(* Schneider Machine Expert - Basic project laba2, file version 2.4.0.0 *)
(* ProjectInformations: Name=New project *)

HARDWARE
  Cpu 0: TM221C16T
  Cartridge1 0: TMC2AQ2V
  EthernetConfiguration: NetworkName=M221, IpAllocationMode=FixedAddress, IpAddress=0.0.0.0, SubnetMask=0.0.0.0
  EthernetConfiguration: NetworkName=M221, IpAllocationMode=FixedAddress, IpAddress=0.0.0.0, SubnetMask=0.0.0.0
  SerialLineConfiguration: Baud=Baud19200, Parity=ParityEven, DataBits=DataBits8, StopBits=StopBits1, PhysicalMedium=PhysicalMediumRs485, TransmissionMode=TransmissionModeModbusRtu, SlaveId=1, Addressing=SlaveAddressing
  MastTask: UsePeriodScanMode=false, PeriodScan=100
  FastTask: Period=255
  CpuBehavior: StartingMode=StartAsPreviousState, AutoSaveRamOnEeprom=true, WatchdogPeriod=250

SYMBOLS  (address, symbol, comment, settings)
  %M100     S_IDLE
  %M101     S_LOAD1
  %M102     S_LOAD2
  %M103     S_HEA1
  %M104     S_HEA2
  %M105     S_DWNLD
  %S13      SB_FIRSTRUN  "Indicates the first controller cycle in RUN mode"
  %I0.0     SB1_PUSK
  %I0.1     SB2_STOP
  %I0.2     LS1_LO
  %I0.3     LS2_MD
  %I0.4     LS3_HI
  %Q0.0     LVS1
  %Q0.1     LVS2
  %Q0.2     LVS3
  %IW0.0    TE1  [Type=Type_0_10V, Scope=Scope_Normal, Minimum=0, Maximum=1000]
  %QW0.100  TV1  [Type=Type_0_10V, Scope=Scope_Customized, Minimum=0, Maximum=10000]

POU New POU
  (* SectionNumber=1 *)

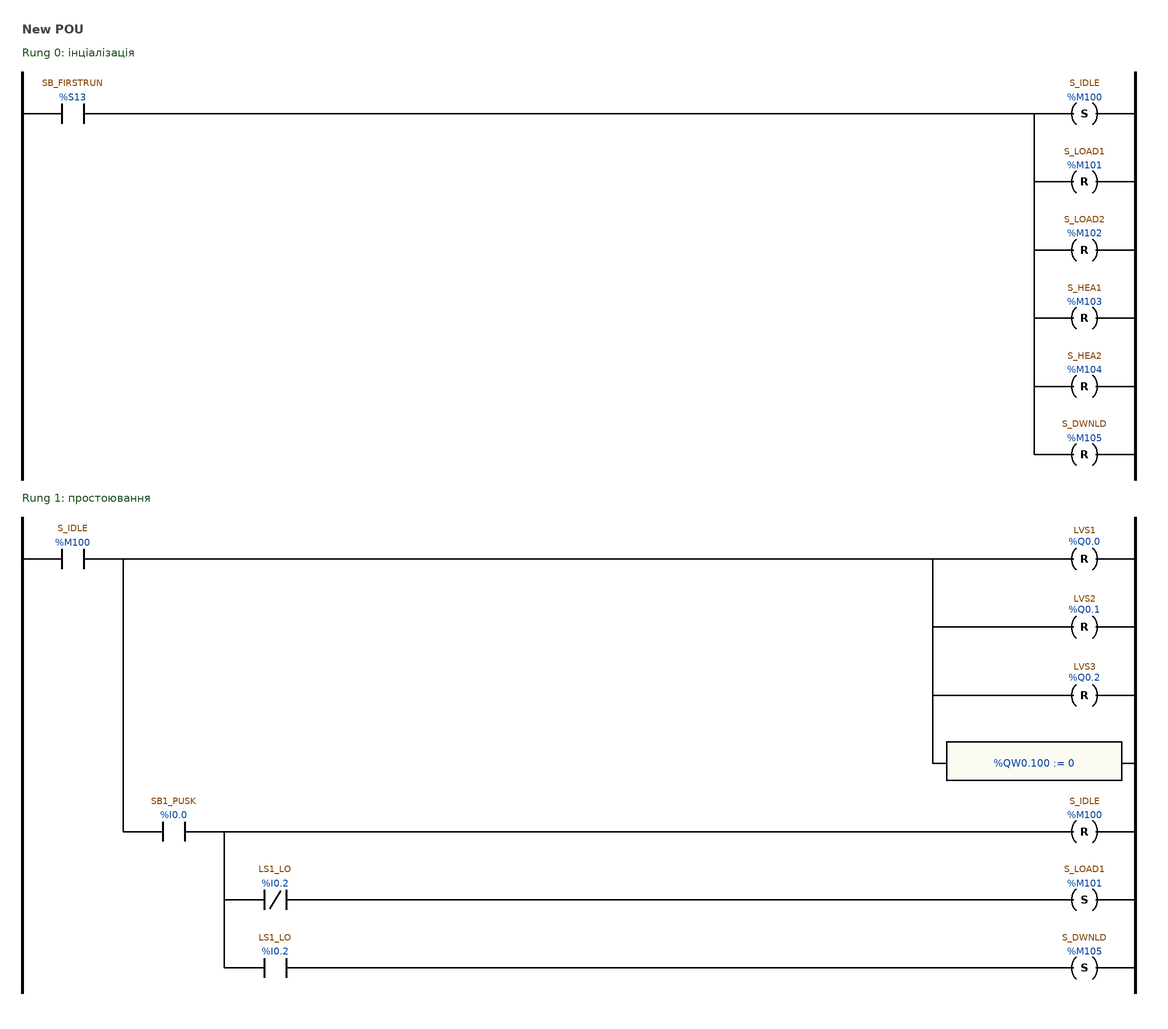

// Rung 0: інціалізація
  LD %S13                 (* SB_FIRSTRUN *)
  S %M100                 (* S_IDLE *)
  R %M101                 (* S_LOAD1 *)
  R %M102                 (* S_LOAD2 *)
  R %M103                 (* S_HEA1 *)
  R %M104                 (* S_HEA2 *)
  R %M105                 (* S_DWNLD *)
  // as ST:
  //   IF SB_FIRSTRUN THEN S_IDLE := TRUE; END_IF;
  //   IF SB_FIRSTRUN THEN S_LOAD1 := FALSE; END_IF;
  //   IF SB_FIRSTRUN THEN S_LOAD2 := FALSE; END_IF;
  //   IF SB_FIRSTRUN THEN S_HEA1 := FALSE; END_IF;
  //   IF SB_FIRSTRUN THEN S_HEA2 := FALSE; END_IF;
  //   IF SB_FIRSTRUN THEN S_DWNLD := FALSE; END_IF;

// Rung 1: простоювання
  LD %M100                (* S_IDLE *)
  MPS
  R %Q0.0                 (* LVS1 *)
  R %Q0.1                 (* LVS2 *)
  R %Q0.2                 (* LVS3 *)
  [ %QW0.100 := 0 ]       (* TV1 *)
  MPP
  AND %I0.0               (* SB1_PUSK *)
  MPS
  R %M100                 (* S_IDLE *)
  MRD
  ANDN %I0.2              (* LS1_LO *)
  S %M101                 (* S_LOAD1 *)
  MPP
  AND %I0.2               (* LS1_LO *)
  S %M105                 (* S_DWNLD *)
  // as ST:
  //   IF S_IDLE THEN LVS1 := FALSE; END_IF;
  //   IF S_IDLE THEN LVS2 := FALSE; END_IF;
  //   IF S_IDLE THEN LVS3 := FALSE; END_IF;
  //   IF S_IDLE THEN TV1 := 0; END_IF;
  //   _t1 := S_IDLE AND SB1_PUSK;
  //   IF _t1 THEN S_IDLE := FALSE; END_IF;
  //   IF _t1 AND NOT LS1_LO THEN S_LOAD1 := TRUE; END_IF;
  //   IF _t1 AND LS1_LO THEN S_DWNLD := TRUE; END_IF;

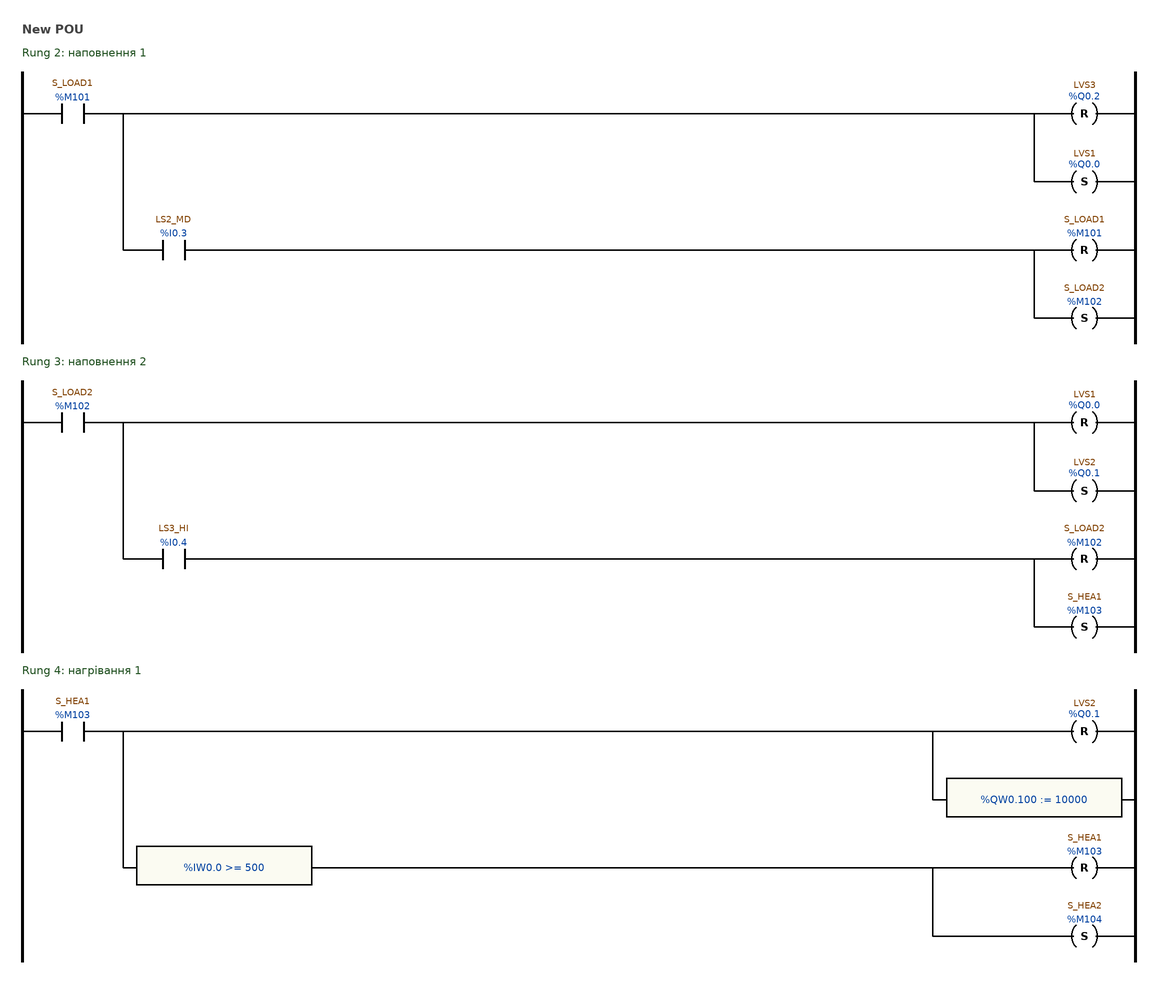

// Rung 2: наповнення 1
  LD %M101                (* S_LOAD1 *)
  MPS
  R %Q0.2                 (* LVS3 *)
  S %Q0.0                 (* LVS1 *)
  MPP
  AND %I0.3               (* LS2_MD *)
  R %M101                 (* S_LOAD1 *)
  S %M102                 (* S_LOAD2 *)
  // as ST:
  //   IF S_LOAD1 THEN LVS3 := FALSE; END_IF;
  //   IF S_LOAD1 THEN LVS1 := TRUE; END_IF;
  //   _t1 := S_LOAD1 AND LS2_MD;
  //   IF _t1 THEN S_LOAD1 := FALSE; END_IF;
  //   IF _t1 THEN S_LOAD2 := TRUE; END_IF;

// Rung 3: наповнення 2
  LD %M102                (* S_LOAD2 *)
  MPS
  R %Q0.0                 (* LVS1 *)
  S %Q0.1                 (* LVS2 *)
  MPP
  AND %I0.4               (* LS3_HI *)
  R %M102                 (* S_LOAD2 *)
  S %M103                 (* S_HEA1 *)
  // as ST:
  //   IF S_LOAD2 THEN LVS1 := FALSE; END_IF;
  //   IF S_LOAD2 THEN LVS2 := TRUE; END_IF;
  //   _t1 := S_LOAD2 AND LS3_HI;
  //   IF _t1 THEN S_LOAD2 := FALSE; END_IF;
  //   IF _t1 THEN S_HEA1 := TRUE; END_IF;

// Rung 4: нагрівання 1
  LD %M103                (* S_HEA1 *)
  MPS
  R %Q0.1                 (* LVS2 *)
  [ %QW0.100 := 10000 ]   (* TV1 *)
  MPP
  AND [ %IW0.0 >= 500 ]   (* TE1 *)
  R %M103                 (* S_HEA1 *)
  S %M104                 (* S_HEA2 *)
  // as ST:
  //   IF S_HEA1 THEN LVS2 := FALSE; END_IF;
  //   IF S_HEA1 THEN TV1 := 10000; END_IF;
  //   _t1 := S_HEA1 AND TE1 >= 500;
  //   IF _t1 THEN S_HEA1 := FALSE; END_IF;
  //   IF _t1 THEN S_HEA2 := TRUE; END_IF;

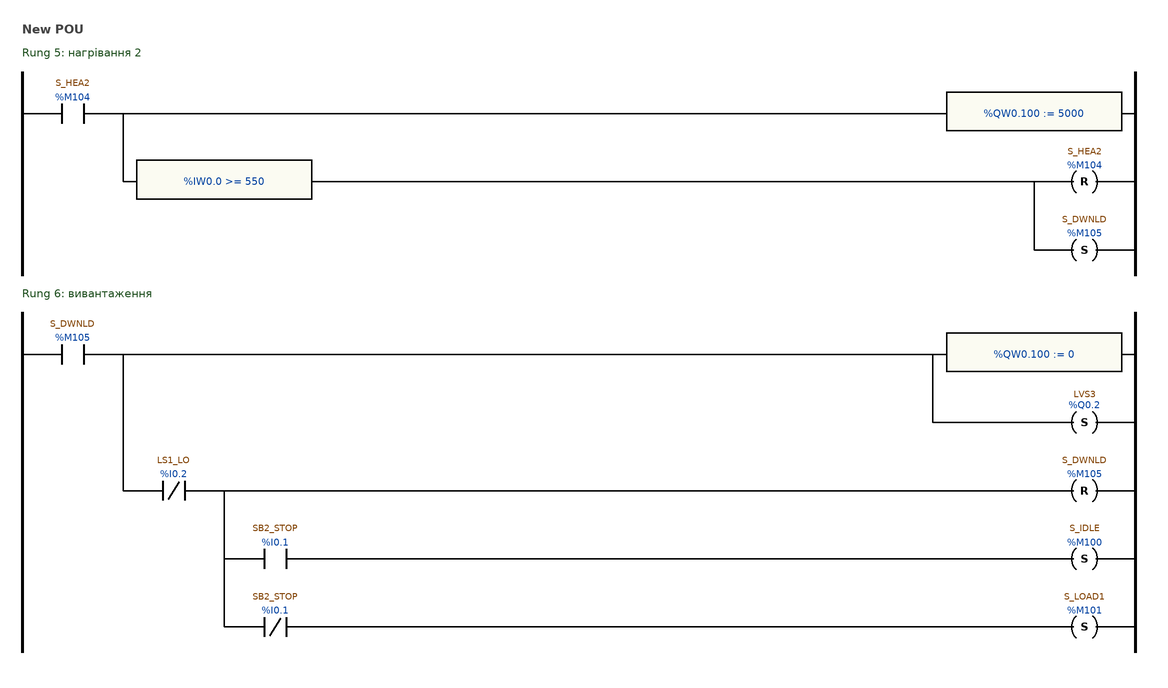

// Rung 5: нагрівання 2
  LD %M104                (* S_HEA2 *)
  MPS
  [ %QW0.100 := 5000 ]    (* TV1 *)
  MPP
  AND [ %IW0.0 >= 550 ]   (* TE1 *)
  R %M104                 (* S_HEA2 *)
  S %M105                 (* S_DWNLD *)
  // as ST:
  //   IF S_HEA2 THEN TV1 := 5000; END_IF;
  //   _t1 := S_HEA2 AND TE1 >= 550;
  //   IF _t1 THEN S_HEA2 := FALSE; END_IF;
  //   IF _t1 THEN S_DWNLD := TRUE; END_IF;

// Rung 6: вивантаження
  LD %M105                (* S_DWNLD *)
  MPS
  [ %QW0.100 := 0 ]       (* TV1 *)
  S %Q0.2                 (* LVS3 *)
  MPP
  ANDN %I0.2              (* LS1_LO *)
  MPS
  R %M105                 (* S_DWNLD *)
  MRD
  AND %I0.1               (* SB2_STOP *)
  S %M100                 (* S_IDLE *)
  MPP
  ANDN %I0.1              (* SB2_STOP *)
  S %M101                 (* S_LOAD1 *)
  // as ST:
  //   IF S_DWNLD THEN TV1 := 0; END_IF;
  //   IF S_DWNLD THEN LVS3 := TRUE; END_IF;
  //   _t1 := S_DWNLD AND NOT LS1_LO;
  //   IF _t1 THEN S_DWNLD := FALSE; END_IF;
  //   IF _t1 AND SB2_STOP THEN S_IDLE := TRUE; END_IF;
  //   IF _t1 AND NOT SB2_STOP THEN S_LOAD1 := TRUE; END_IF;
